// Mitsubishi GX Works2 project: ServoConveyor   PLC: Q03UD

PROGRAM MAIN
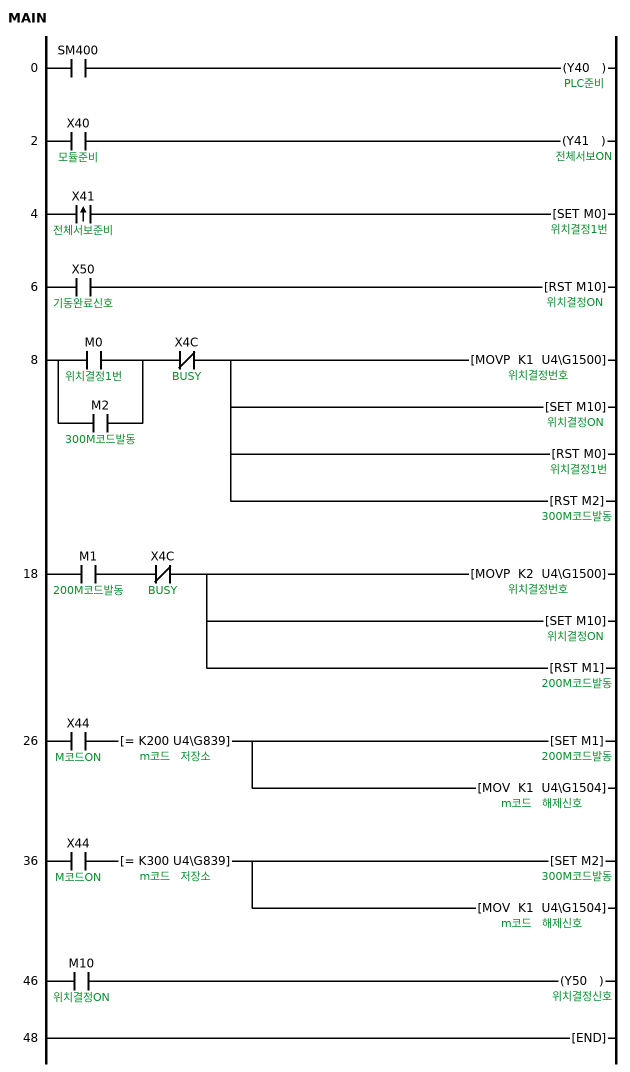
0     LD      SM400
      OUT     Y40  ; PLC준비
2     LD      X40  ; 모듈준비
      OUT     Y41  ; 전체서보ON
4     LDP     X41  ; 전체서보준비
      SET     M0  ; 위치결정1번
6     LD      X50  ; 기동완료신호
      RST     M10  ; 위치결정ON
8     LD      M0  ; 위치결정1번
      OR      M2  ; 300M코드발동
      ANI     X4C  ; BUSY
      MOVP    K1 U4\G1500  ; 위치결정번호
      SET     M10  ; 위치결정ON
      RST     M0  ; 위치결정1번
      RST     M2  ; 300M코드발동
18    LD      M1  ; 200M코드발동
      ANI     X4C  ; BUSY
      MOVP    K2 U4\G1500
      SET     M10  ; 위치결정ON
      RST     M1  ; 200M코드발동
26    LD      X44  ; M코드ON
      AND=    K200 U4\G839  ; m코드   저장소
      SET     M1  ; 200M코드발동
      MOV     K1 U4\G1504  ; m코드   해제신호
36    LD      X44  ; M코드ON
      AND=    K300 U4\G839  ; m코드   저장소
      SET     M2  ; 300M코드발동
      MOV     K1 U4\G1504
46    LD      M10  ; 위치결정ON
      OUT     Y50  ; 위치결정신호
48    END
END_PROGRAM

PROGRAM IOCHECK
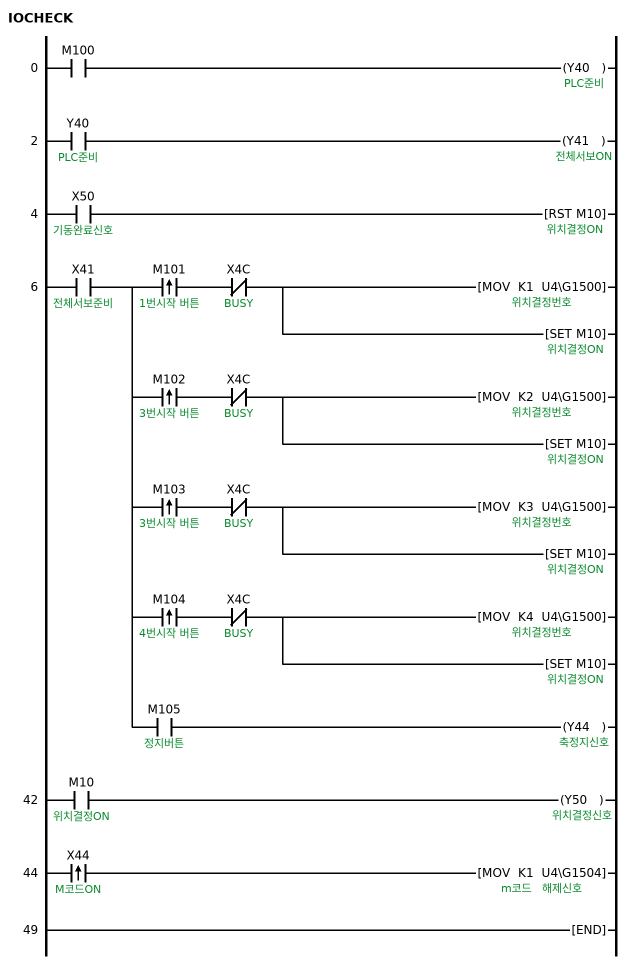
0     LD      M100
      OUT     Y40  ; PLC준비
2     LD      Y40  ; PLC준비
      OUT     Y41  ; 전체서보ON
4     LD      X50  ; 기동완료신호
      RST     M10  ; 위치결정ON
6     LD      X41  ; 전체서보준비
      MPS
      ANDP    M101  ; 1번시작 버튼
      ANI     X4C  ; BUSY
      MOV     K1 U4\G1500  ; 위치결정번호
      SET     M10  ; 위치결정ON
      MRD
      ANDP    M102  ; 3번시작 버튼
      ANI     X4C  ; BUSY
      MOV     K2 U4\G1500
      SET     M10  ; 위치결정ON
      MRD
      ANDP    M103  ; 3번시작 버튼
      ANI     X4C  ; BUSY
      MOV     K3 U4\G1500
      SET     M10  ; 위치결정ON
      MRD
      ANDP    M104  ; 4번시작 버튼
      ANI     X4C  ; BUSY
      MOV     K4 U4\G1500
      SET     M10  ; 위치결정ON
      MPP
      AND     M105  ; 정지버튼
      OUT     Y44  ; 축정지신호
42    LD      M10  ; 위치결정ON
      OUT     Y50  ; 위치결정신호
44    LDP     X44  ; M코드ON
      MOV     K1 U4\G1504  ; m코드   해제신호
49    END
END_PROGRAM

// device comments not shown above
M40  ; 모듈준비
